{attribute 'GeneratedUsingTerminal: IL2300-B110-0017'}
{attribute addProperty BoxType "IL2300-B110-0017"}
{attribute addProperty Id "Term_20KL_D4CFBC220Term_391_Ix1000KL_8EF4D3E90"}
{attribute addProperty CRC "2349215268"}
{attribute addProperty Size "0"}
TYPE A_0020_IL2300_B110_0017_8C062E24 EXTENDS IL2300_13409EDF :
STRUCT
	{attribute addProperty Name "Term_20"}
	Term_20 : KL_D4CFBC22;
	{attribute addProperty Name "Term_391_Ix1000"}
	Term_391_Ix1000 : KL_8EF4D3E9;
END_STRUCT
END_TYPE

(* stored: Version 1.2.0.0, ProductVersion 3.1.4024.9
   DUT A_0020_IL2300_B110_0017_8C062E24: Id {0308b1f0-08f8-4260-a664-f4d02ede0bf6} *)
